# EPICS autosave request: iocBoot/ioc13lab_linux/auto_settings.req
file "calc_GSECARS.req",                P=$(P)
file "Galil_settings.req",              P=$(P)
#file "XPS_settings.req",                P=$(P)
